(* IEC 61131-3 sources: ServoDriveControllerCode_Gen3SOScompressor/src/DUT, 7 files *)

(* ---- DataTypes.st ---- *)
(* ============================================================================
   DataTypes - All Data Type Definitions

   Project: Gen3 SOS Compressor Servo Controller
   Controller: Yaskawa MP2600iec

   Description:
   Combined data type definitions for the servo controller project.
   Contains all enumerations and structures used throughout the codebase.

   Contents:
   - E_OperatingMode: Operating mode enumeration (3-bit encoding)
   - E_FaultCode: Fault code enumeration (3-bit encoding)
   - E_SystemState: System state machine enumeration
   - ST_AxisLimits: Position, velocity, torque, accel/decel limits
   - ST_HomingParams: Homing sequence parameters
   ============================================================================ *)

(* ============================================================================
   E_OperatingMode - Operating Mode Enumeration

   Encoding:
   - Bits come from DI0 (LSB), DI1, DI2 (MSB)
   - Mode value = DI2*4 + DI1*2 + DI0
   ============================================================================ *)

(* IMPORTANT: Member order defines implicit integer values (0-7).
   These values map to 3-bit mode encoding on DI0-DI2 and DO0-DO2. Do not reorder. *)
TYPE E_OperatingMode :
(
    MODE_IDLE,               (* implicit 0 - 000: Idle - Drive OFF, brake engaged *)
    MODE_BRAKE_HOLD,         (* implicit 1 - 001: Brake Hold - Drive ON, brake engaged *)
    MODE_POSITION,           (* implicit 2 - 010: Position Control - Analog reference *)
    MODE_VELOCITY,           (* implicit 3 - 011: Velocity Control - Analog reference *)
    MODE_TORQUE,             (* implicit 4 - 100: Torque Control - Analog reference *)
    MODE_GO_HOME,            (* implicit 5 - 101: Go Home - Move to home position *)
    MODE_HOME_LIMIT,         (* implicit 6 - 110: Home to Limit Switch *)
    MODE_HOME_EOT            (* implicit 7 - 111: Home to End-of-Travel (torque detection) *)
);
END_TYPE;

(* ============================================================================
   E_FaultCode - Fault Code Enumeration

   When doFaultActive is HIGH, the 3-bit fault code is output on DO0-DO2
   instead of mode confirmation.

   Encoding:
   - DO0 = bit 0 (LSB), DO1 = bit 1, DO2 = bit 2 (MSB)
   - Fault value = DO2*4 + DO1*2 + DO0
   ============================================================================ *)

(* IMPORTANT: Member order defines implicit integer values (0-7).
   These values map to 3-bit fault codes on DO0-DO2. Do not reorder. *)
TYPE E_FaultCode :
(
    FAULT_NONE,              (* implicit 0 - 000: No fault / fault cleared *)
    FAULT_HANDSHAKE,         (* implicit 1 - 001: Handshake timeout or mismatch *)
    FAULT_DRIVE,             (* implicit 2 - 010: Drive fault (from servo amplifier) *)
    FAULT_POSITION,          (* implicit 3 - 011: Position limit exceeded *)
    FAULT_HOMING_REQ,        (* implicit 4 - 100: Homing requirement not met *)
    FAULT_PISTON_EXIT,       (* implicit 5 - 101: Piston exit prevention triggered *)
    FAULT_LIMIT_SWITCH,      (* implicit 6 - 110: Limit switch fault *)
    FAULT_ENCODER            (* implicit 7 - 111: Encoder / absolute position fault *)
);
END_TYPE;

(* ============================================================================
   E_SystemState - System State Enumeration

   All possible states in the main state machine. States are grouped by
   function: Initialization, Idle, Transitions, Operational, and Fault states.
   ============================================================================ *)

(* NOTE: Implicit integer values do not matter for this enum.
   All code references states by name, never by numeric value.
   States are grouped logically below for readability. *)
TYPE E_SystemState :
(
    (* Initialization States *)
    ST_INIT,                 (* Power-on initialization *)
    ST_ENCODER_CHECK,        (* Validate absolute encoder status *)
    ST_REQUIRE_ABS_HOME,     (* Encoder invalid, set flag and proceed to idle *)

    (* Idle State *)
    ST_IDLE,                 (* Drive OFF, brake engaged, awaiting commands *)

    (* Transition States - Activation *)
    ST_DRIVE_ENABLE,         (* Power on drive, wait for ready *)
    ST_BRAKE_RELEASE,        (* Release brake, wait for mechanical delay *)

    (* Operational States *)
    ST_BRAKE_HOLD,           (* Mode 001: Drive ON, brake engaged *)
    ST_POSITION_CTRL,        (* Mode 010: Position control active *)
    ST_VELOCITY_CTRL,        (* Mode 011: Velocity control active *)
    ST_TORQUE_CTRL,          (* Mode 100: Torque control active *)
    ST_GO_HOME,              (* Mode 101: Moving to home position *)

    (* Homing States *)
    ST_HOME_LIMIT,           (* Mode 110: Homing to limit switch - uses FB_HomeLimit *)
    ST_HOME_EOT,             (* Mode 111: Homing to end-of-travel - uses FB_HomeEOT *)
    ST_HOME_COMPLETE,        (* Homing finished, awaiting mode change *)

    (* DEPRECATED: Homing sub-states - Limit Switch (Mode 110)
       These states are now handled internally by FB_HomeLimit. *)
    ST_HOME_LIM_APPROACH,    (* DEPRECATED - use FB_HomeLimit *)
    ST_HOME_LIM_DETECT,      (* DEPRECATED - use FB_HomeLimit *)
    ST_HOME_LIM_BACKOFF,     (* DEPRECATED - use FB_HomeLimit *)
    ST_HOME_LIM_SETREF,      (* DEPRECATED - use FB_HomeLimit *)

    (* DEPRECATED: Homing sub-states - End-of-Travel (Mode 111)
       These states are now handled internally by FB_HomeEOT. *)
    ST_HOME_EOT_FAST,        (* DEPRECATED - use FB_HomeEOT *)
    ST_HOME_EOT_SLOW,        (* DEPRECATED - use FB_HomeEOT *)
    ST_HOME_EOT_DETECT,      (* DEPRECATED - use FB_HomeEOT *)
    ST_HOME_EOT_SETREF,      (* DEPRECATED - use FB_HomeEOT *)

    (* Transition State - Inter-Mode *)
    ST_HOLD_POSITION,        (* MC_Halt active, brake disengaged, awaiting handshake *)

    (* Transition States - Deactivation *)
    ST_BRAKE_ENGAGE,         (* Engage brake, wait for mechanical delay *)
    ST_DRIVE_DISABLE,        (* Power off drive, return to idle *)

    (* Fault States *)
    ST_FAULT,                (* Fault active, no brake, MC_Halt, await handshake/timeout *)
    ST_FAULT_RECOVERY,       (* Legacy - may be removed *)
    ST_FAULT_IDLE            (* Drive disabled, brake engaged, await fault reset handshake *)
);
END_TYPE;

(* ============================================================================
   ST_AxisLimits - Axis Limits Structure

   Structure containing position, velocity, and torque limits.
   Used for mode-dependent limit configuration.
   ============================================================================ *)

TYPE ST_AxisLimits :
STRUCT
    (* Position limits (mm) *)
    PosMax          : LREAL;    (* Maximum position limit *)
    PosMin          : LREAL;    (* Minimum position limit *)

    (* Velocity limits (mm/s) *)
    VelMax          : LREAL;    (* Maximum velocity limit *)
    VelMin          : LREAL;    (* Minimum velocity limit (usually negative of VelMax) *)

    (* Torque limits (% of rated) *)
    TorqueMax       : LREAL;    (* Maximum torque limit (positive direction) *)
    TorqueMin       : LREAL;    (* Minimum torque limit (negative direction) *)

    (* Acceleration/Deceleration limits (mm/s^2) *)
    AccelMax        : LREAL;    (* Maximum acceleration *)
    DecelMax        : LREAL;    (* Maximum deceleration *)
END_STRUCT;
END_TYPE;

(* ============================================================================
   ST_HomingParams - Homing Parameters Structure

   Structure containing parameters for homing sequences.
   Supports both limit switch homing (Mode 110) and EOT homing (Mode 111).
   ============================================================================ *)

TYPE ST_HomingParams :
STRUCT
    (* Approach velocities (mm/s) *)
    VelFast         : LREAL;    (* Fast approach velocity *)
    VelSlow         : LREAL;    (* Slow approach velocity *)

    (* Torque parameters (% of rated) *)
    TorqueThreshold : LREAL;    (* Stall detection threshold (EOT homing) *)
    TorqueLimit     : LREAL;    (* Torque limit during slow approach *)

    (* Distance parameters (mm) *)
    ApproachDist    : LREAL;    (* Distance for slow approach phase *)
    BackoffDist     : LREAL;    (* Distance to back off after detection *)

    (* Position to set after homing (mm) *)
    SetPosition     : LREAL;    (* Position value to assign at home point *)

    (* Timing *)
    StallDetectTime : TIME;     (* Time to confirm stall condition *)
    Timeout         : TIME;     (* Overall homing sequence timeout *)

    (* Direction *)
    Direction       : INT;      (* Homing direction: 1 = positive, -1 = negative *)
END_STRUCT;
END_TYPE;

(* ---- E_FaultCode.st ---- *)
(* ============================================================================
   E_FaultCode - Fault Code Enumeration

   Project: Gen3 SOS Compressor Servo Controller
   Controller: Yaskawa MP2600iec

   Description:
   Enumeration of fault codes. When doFaultActive is HIGH, the 3-bit fault
   code is output on DO0-DO2 instead of mode confirmation.

   Encoding:
   - DO0 = bit 0 (LSB), DO1 = bit 1, DO2 = bit 2 (MSB)
   - Fault value = DO2*4 + DO1*2 + DO0
   ============================================================================ *)

TYPE E_FaultCode :
(
    FAULT_NONE := 0,            (* 000: No fault / fault cleared *)
    FAULT_HANDSHAKE := 1,       (* 001: Handshake timeout or mismatch *)
    FAULT_DRIVE := 2,           (* 010: Drive fault (from servo amplifier) *)
    FAULT_POSITION := 3,        (* 011: Position limit exceeded *)
    FAULT_HOMING_REQ := 4,      (* 100: Homing requirement not met *)
    FAULT_PISTON_EXIT := 5,     (* 101: Piston exit prevention triggered *)
    FAULT_LIMIT_SWITCH := 6,    (* 110: Limit switch fault *)
    FAULT_ENCODER := 7          (* 111: Encoder / absolute position fault *)
);
END_TYPE

(* ---- E_OperatingMode.st ---- *)
(* ============================================================================
   E_OperatingMode - Operating Mode Enumeration

   Project: Gen3 SOS Compressor Servo Controller
   Controller: Yaskawa MP2600iec

   Description:
   Enumeration of operating modes corresponding to the 3-bit mode encoding
   from the master controller.

   Encoding:
   - Bits come from DI0 (LSB), DI1, DI2 (MSB)
   - Mode value = DI2*4 + DI1*2 + DI0
   ============================================================================ *)

TYPE E_OperatingMode :
(
    MODE_IDLE := 0,             (* 000: Idle - Drive OFF, brake engaged *)
    MODE_BRAKE_HOLD := 1,       (* 001: Brake Hold - Drive ON, brake engaged *)
    MODE_POSITION := 2,         (* 010: Position Control - Analog reference *)
    MODE_VELOCITY := 3,         (* 011: Velocity Control - Analog reference *)
    MODE_TORQUE := 4,           (* 100: Torque Control - Analog reference *)
    MODE_GO_HOME := 5,          (* 101: Go Home - Move to home position *)
    MODE_HOME_LIMIT := 6,       (* 110: Home to Limit Switch *)
    MODE_HOME_EOT := 7          (* 111: Home to End-of-Travel (torque detection) *)
);
END_TYPE

(* ---- E_SystemState.st ---- *)
(* ============================================================================
   E_SystemState - System State Enumeration

   Project: Gen3 SOS Compressor Servo Controller
   Controller: Yaskawa MP2600iec

   Description:
   Enumeration of all possible states in the main state machine.
   States are grouped by function: Initialization, Idle, Transitions,
   Operational, and Fault states.
   ============================================================================ *)

TYPE E_SystemState :
(
    (* ========================================================================
       INITIALIZATION STATES (0-9)
       ======================================================================== *)
    ST_INIT := 0,               (* Power-on initialization *)
    ST_ENCODER_CHECK := 1,      (* Validate absolute encoder status *)
    ST_REQUIRE_ABS_HOME := 2,   (* Encoder invalid, set flag and proceed to idle *)

    (* ========================================================================
       IDLE STATE (10-19)
       ======================================================================== *)
    ST_IDLE := 10,              (* Drive OFF, brake engaged, awaiting commands *)

    (* ========================================================================
       TRANSITION STATES - ACTIVATION (20-29)
       ======================================================================== *)
    ST_DRIVE_ENABLE := 20,      (* Power on drive, wait for ready *)
    ST_BRAKE_RELEASE := 21,     (* Release brake, wait for mechanical delay *)

    (* ========================================================================
       OPERATIONAL STATES (30-59)
       ======================================================================== *)
    ST_BRAKE_HOLD := 30,        (* Mode 001: Drive ON, brake engaged *)
    ST_POSITION_CTRL := 31,     (* Mode 010: Position control active *)
    ST_VELOCITY_CTRL := 32,     (* Mode 011: Velocity control active *)
    ST_TORQUE_CTRL := 33,       (* Mode 100: Torque control active *)
    ST_GO_HOME := 34,           (* Mode 101: Moving to home position *)

    (* Homing states *)
    ST_HOME_LIMIT := 40,        (* Mode 110: Homing to limit switch - uses FB_HomeLimit *)
    ST_HOME_EOT := 41,          (* Mode 111: Homing to end-of-travel - uses FB_HomeEOT *)
    ST_HOME_COMPLETE := 42,     (* Homing finished, awaiting mode change *)

    (* DEPRECATED: Homing sub-states - Limit Switch (Mode 110)
       These states are now handled internally by FB_HomeLimit.
       Values kept for backward compatibility - states redirect to ST_HOME_LIMIT. *)
    ST_HOME_LIM_APPROACH := 43, (* DEPRECATED - use FB_HomeLimit *)
    ST_HOME_LIM_DETECT := 44,   (* DEPRECATED - use FB_HomeLimit *)
    ST_HOME_LIM_BACKOFF := 45,  (* DEPRECATED - use FB_HomeLimit *)
    ST_HOME_LIM_SETREF := 46,   (* DEPRECATED - use FB_HomeLimit *)

    (* DEPRECATED: Homing sub-states - End-of-Travel (Mode 111)
       These states are now handled internally by FB_HomeEOT.
       Values kept for backward compatibility - states redirect to ST_HOME_EOT. *)
    ST_HOME_EOT_FAST := 50,     (* DEPRECATED - use FB_HomeEOT *)
    ST_HOME_EOT_SLOW := 51,     (* DEPRECATED - use FB_HomeEOT *)
    ST_HOME_EOT_DETECT := 52,   (* DEPRECATED - use FB_HomeEOT *)
    ST_HOME_EOT_SETREF := 53,   (* DEPRECATED - use FB_HomeEOT *)

    (* ========================================================================
       TRANSITION STATE - INTER-MODE (60-69)
       ======================================================================== *)
    ST_HOLD_POSITION := 60,     (* MC_Halt active, brake disengaged, awaiting handshake *)

    (* ========================================================================
       TRANSITION STATES - DEACTIVATION (70-79)
       ======================================================================== *)
    ST_BRAKE_ENGAGE := 70,      (* Engage brake, wait for mechanical delay *)
    ST_DRIVE_DISABLE := 71,     (* Power off drive, return to idle *)

    (* ========================================================================
       FAULT STATES (90-99)
       ======================================================================== *)
    ST_FAULT := 90,             (* Fault active, no brake, MC_Halt, await handshake/timeout *)
    ST_FAULT_RECOVERY := 91,    (* Legacy - may be removed *)
    ST_FAULT_IDLE := 92         (* Drive disabled, brake engaged, await fault reset handshake *)

);
END_TYPE

(* ---- ST_AxisLimits.st ---- *)
(* ============================================================================
   ST_AxisLimits - Axis Limits Structure

   Project: Gen3 SOS Compressor Servo Controller
   Controller: Yaskawa MP2600iec

   Description:
   Structure containing position, velocity, and torque limits.
   Used for mode-dependent limit configuration.
   ============================================================================ *)

TYPE ST_AxisLimits :
STRUCT
    (* Position limits (mm) *)
    PosMax          : LREAL;    (* Maximum position limit *)
    PosMin          : LREAL;    (* Minimum position limit *)

    (* Velocity limits (mm/s) *)
    VelMax          : LREAL;    (* Maximum velocity limit *)
    VelMin          : LREAL;    (* Minimum velocity limit (usually negative of VelMax) *)

    (* Torque limits (% of rated) *)
    TorqueMax       : LREAL;    (* Maximum torque limit (positive direction) *)
    TorqueMin       : LREAL;    (* Minimum torque limit (negative direction) *)

    (* Acceleration/Deceleration limits (mm/s^2) *)
    AccelMax        : LREAL;    (* Maximum acceleration *)
    DecelMax        : LREAL;    (* Maximum deceleration *)
END_STRUCT
END_TYPE

(* ---- ST_HomingParams.st ---- *)
(* ============================================================================
   ST_HomingParams - Homing Parameters Structure

   Project: Gen3 SOS Compressor Servo Controller
   Controller: Yaskawa MP2600iec

   Description:
   Structure containing parameters for homing sequences.
   Supports both limit switch homing (Mode 110) and EOT homing (Mode 111).
   ============================================================================ *)

TYPE ST_HomingParams :
STRUCT
    (* Approach velocities (mm/s) *)
    VelFast         : LREAL;    (* Fast approach velocity *)
    VelSlow         : LREAL;    (* Slow approach velocity *)

    (* Torque parameters (% of rated) *)
    TorqueThreshold : LREAL;    (* Stall detection threshold (EOT homing) *)
    TorqueLimit     : LREAL;    (* Torque limit during slow approach *)

    (* Distance parameters (mm) *)
    ApproachDist    : LREAL;    (* Distance for slow approach phase *)
    BackoffDist     : LREAL;    (* Distance to back off after detection *)

    (* Position to set after homing (mm) *)
    SetPosition     : LREAL;    (* Position value to assign at home point *)

    (* Timing *)
    StallDetectTime : TIME;     (* Time to confirm stall condition *)
    Timeout         : TIME;     (* Overall homing sequence timeout *)

    (* Direction *)
    Direction       : INT;      (* Homing direction: 1 = positive, -1 = negative *)
END_STRUCT
END_TYPE

(* ---- EnumConversions.st ---- *)
(* ============================================================================
   EnumConversions - Centralized Enum Conversion Functions

   Project: Gen3 SOS Compressor Servo Controller
   Controller: Yaskawa MP2600iec

   Description:
   Centralized functions for converting between enumerations and their
   integer/bit representations. All enum conversion logic should be here
   to ensure consistency across the codebase.
   ============================================================================ *)

(* ============================================================================
   MODE CONVERSIONS
   ============================================================================ *)

(* Convert E_OperatingMode to integer value (0-7) *)
FUNCTION ModeToInt : INT
VAR_INPUT
    Mode : E_OperatingMode;
END_VAR

CASE Mode OF
    MODE_IDLE:       ModeToInt := 0;
    MODE_BRAKE_HOLD: ModeToInt := 1;
    MODE_POSITION:   ModeToInt := 2;
    MODE_VELOCITY:   ModeToInt := 3;
    MODE_TORQUE:     ModeToInt := 4;
    MODE_GO_HOME:    ModeToInt := 5;
    MODE_HOME_LIMIT: ModeToInt := 6;
    MODE_HOME_EOT:   ModeToInt := 7;
ELSE
    ModeToInt := 0;
END_CASE

END_FUNCTION

(* Convert integer value (0-7) to E_OperatingMode *)
FUNCTION IntToMode : E_OperatingMode
VAR_INPUT
    Value : INT;
END_VAR

CASE Value OF
    0: IntToMode := MODE_IDLE;
    1: IntToMode := MODE_BRAKE_HOLD;
    2: IntToMode := MODE_POSITION;
    3: IntToMode := MODE_VELOCITY;
    4: IntToMode := MODE_TORQUE;
    5: IntToMode := MODE_GO_HOME;
    6: IntToMode := MODE_HOME_LIMIT;
    7: IntToMode := MODE_HOME_EOT;
ELSE
    IntToMode := MODE_IDLE;
END_CASE

END_FUNCTION

(* Convert 3 digital input bits to E_OperatingMode *)
FUNCTION BitsToMode : E_OperatingMode
VAR_INPUT
    Bit0 : BOOL;    (* LSB *)
    Bit1 : BOOL;
    Bit2 : BOOL;    (* MSB *)
END_VAR
VAR
    nValue : INT;
END_VAR

nValue := 0;
IF Bit0 THEN nValue := nValue + 1; END_IF
IF Bit1 THEN nValue := nValue + 2; END_IF
IF Bit2 THEN nValue := nValue + 4; END_IF

BitsToMode := IntToMode(nValue);

END_FUNCTION

(* Convert E_OperatingMode to 3 output bits *)
FUNCTION ModeToBits
VAR_INPUT
    Mode : E_OperatingMode;
END_VAR
VAR_OUTPUT
    Bit0 : BOOL;    (* LSB *)
    Bit1 : BOOL;
    Bit2 : BOOL;    (* MSB *)
END_VAR
VAR
    nValue : INT;
END_VAR

nValue := ModeToInt(Mode);
Bit0 := (nValue AND 1) <> 0;
Bit1 := (nValue AND 2) <> 0;
Bit2 := (nValue AND 4) <> 0;

END_FUNCTION

(* ============================================================================
   FAULT CODE CONVERSIONS
   ============================================================================ *)

(* Convert E_FaultCode to integer value (0-7) *)
FUNCTION FaultToInt : INT
VAR_INPUT
    Fault : E_FaultCode;
END_VAR

CASE Fault OF
    FAULT_NONE:         FaultToInt := 0;
    FAULT_HANDSHAKE:    FaultToInt := 1;
    FAULT_DRIVE:        FaultToInt := 2;
    FAULT_POSITION:     FaultToInt := 3;
    FAULT_HOMING_REQ:   FaultToInt := 4;
    FAULT_PISTON_EXIT:  FaultToInt := 5;
    FAULT_LIMIT_SWITCH: FaultToInt := 6;
    FAULT_ENCODER:      FaultToInt := 7;
ELSE
    FaultToInt := 0;
END_CASE

END_FUNCTION

(* Convert integer value (0-7) to E_FaultCode *)
FUNCTION IntToFault : E_FaultCode
VAR_INPUT
    Value : INT;
END_VAR

CASE Value OF
    0: IntToFault := FAULT_NONE;
    1: IntToFault := FAULT_HANDSHAKE;
    2: IntToFault := FAULT_DRIVE;
    3: IntToFault := FAULT_POSITION;
    4: IntToFault := FAULT_HOMING_REQ;
    5: IntToFault := FAULT_PISTON_EXIT;
    6: IntToFault := FAULT_LIMIT_SWITCH;
    7: IntToFault := FAULT_ENCODER;
ELSE
    IntToFault := FAULT_NONE;
END_CASE

END_FUNCTION

(* Convert E_FaultCode to 3 output bits *)
FUNCTION FaultToBits
VAR_INPUT
    Fault : E_FaultCode;
END_VAR
VAR_OUTPUT
    Bit0 : BOOL;    (* LSB *)
    Bit1 : BOOL;
    Bit2 : BOOL;    (* MSB *)
END_VAR
VAR
    nValue : INT;
END_VAR

nValue := FaultToInt(Fault);
Bit0 := (nValue AND 1) <> 0;
Bit1 := (nValue AND 2) <> 0;
Bit2 := (nValue AND 4) <> 0;

END_FUNCTION

(* ============================================================================
   CROSS-TYPE COMPARISONS
   ============================================================================ *)

(* Check if a fault code value matches mode bits (for fault reset mirroring) *)
FUNCTION FaultMatchesModeBits : BOOL
VAR_INPUT
    Fault : E_FaultCode;
    Mode  : E_OperatingMode;
END_VAR

(* Both use 3-bit encoding 0-7, so we just compare integer values *)
FaultMatchesModeBits := (FaultToInt(Fault) = ModeToInt(Mode));

END_FUNCTION
